TYPE E_CFG_UMC :
(
	Standard := 0,
	LenzeFC := 1,
	MAY_E_CFG_UMC
);
END_TYPE

(* stored: Version 1.1.0.1, ProductVersion 3.1.0.26
   DUT E_CFG_UMC: Id {13c27364-c2e6-4822-9f8f-ab42b9793010} *)
